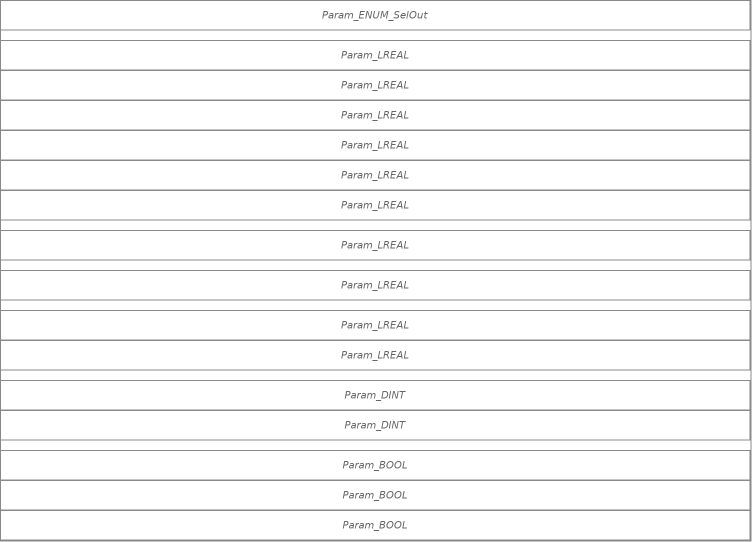
VISUALIZATION Visu_Mparam_Heat  // 752x542
    Frame (0,40 750x30)
        shows Param_LREAL(nIdx := 4)
    Frame (0,70 750x30)
        shows Param_LREAL(nIdx := 6)
    Frame (0,100 750x30)
        shows Param_LREAL(nIdx := 8)
    Frame (0,130 750x30)
        shows Param_LREAL(nIdx := 10)
    Frame (0,380 750x30)
        shows Param_DINT(nIdx := 11)
    Frame (0,0 750x30)
        shows Param_ENUM_SelOut(nIdx := GlobalOne)
    Frame (0,160 750x30)
        shows Param_LREAL(nIdx := 16)
    Frame (0,190 750x30)
        shows Param_LREAL(nIdx := 17)
    Frame (0,230 750x30)
        shows Param_LREAL(nIdx := 21)
    Frame (0,310 750x30)
        shows Param_LREAL(nIdx := 37)
    Frame (0,340 750x30)
        shows Param_LREAL(nIdx := 38)
    Frame (0,450 750x30)
        shows Param_BOOL(nIdx := GlobalOne)
    Frame (0,480 750x30)
        shows Param_BOOL(nIdx := 3)
    Frame (0,510 750x30)
        shows Param_BOOL(nIdx := 18)
    Frame (0,270 750x30)
        shows Param_LREAL(nIdx := 32)
    Frame (0,410 750x30)
        shows Param_DINT(nIdx := 12)
END_VISUALIZATION

(* stored: Version 1.1.0.1, ProductVersion 3.1.4024.12
   Visu Visu_Mparam_Heat: Id {4f578426-2293-467e-8b91-0f0781ab1583} *)
